TYPE "TExtEncoder_Ctrl"
VERSION : 0.1
// Block: TExtEncoder_Ctrl
   STRUCT
      Rst : Bool;
      Home : Bool;
      HomeMode : Int;
      HomePosition : LReal;
   END_STRUCT;

END_TYPE
